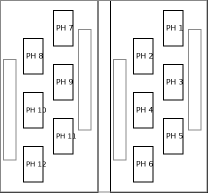
VISUALIZATION VISU_PhEnable_M2  // 208x193
    RoundedRectangle (0,0 98x193)
        toggle PRG_PRINT.sAdsPrintGroup[2].bI_Enable
    Rectangle (53,10 20x36), colour toggle: PRG_PRINT.sAdsPrintHead[7].bI_Enable
        toggle PRG_PRINT.sAdsPrintHead[7].bI_Enable
    Rectangle (23,38 20x36), colour toggle: PRG_PRINT.sAdsPrintHead[8].bI_Enable
        toggle PRG_PRINT.sAdsPrintHead[8].bI_Enable
    Rectangle (53,64 20x36), colour toggle: PRG_PRINT.sAdsPrintHead[9].bI_Enable
        toggle PRG_PRINT.sAdsPrintHead[9].bI_Enable
    Rectangle (23,92 20x36), colour toggle: PRG_PRINT.sAdsPrintHead[10].bI_Enable
        toggle PRG_PRINT.sAdsPrintHead[10].bI_Enable
    Rectangle (53,118 20x36), colour toggle: PRG_PRINT.sAdsPrintHead[11].bI_Enable
        toggle PRG_PRINT.sAdsPrintHead[11].bI_Enable
    Rectangle (23,146 20x36), colour toggle: PRG_PRINT.sAdsPrintHead[12].bI_Enable
        toggle PRG_PRINT.sAdsPrintHead[12].bI_Enable
    Rectangle (15,46 36x20), angle 270, "PH 8", colour toggle: PRG_PRINT.sAdsPrintHead[8].bI_Enable
    Rectangle (45,18 36x20), angle 270, "PH 7", colour toggle: PRG_PRINT.sAdsPrintHead[7].bI_Enable
    Rectangle (45,72 36x20), angle 270, "PH 9", colour toggle: PRG_PRINT.sAdsPrintHead[9].bI_Enable
    Rectangle (15,100 36x20), angle 270, "PH 10", colour toggle: PRG_PRINT.sAdsPrintHead[10].bI_Enable
    Rectangle (45,126 36x20), angle 270, "PH 11", colour toggle: PRG_PRINT.sAdsPrintHead[11].bI_Enable
    Rectangle (15,154 36x20), angle 270, "PH 12", colour toggle: PRG_PRINT.sAdsPrintHead[12].bI_Enable
    Frame (78,29 13x101)
        shows _VISU_PcMiniVertical(m_Inst := PRG_PRINT.FB_PC[3])
    Frame (3,59 13x101)
        shows _VISU_PcMiniVertical(m_Inst := PRG_PRINT.FB_PC[4])
    RoundedRectangle (110,0 98x193)
        toggle PRG_PRINT.sAdsPrintGroup[1].bI_Enable
    Rectangle (163,10 20x36), colour toggle: PRG_PRINT.sAdsPrintHead[1].bI_Enable
        toggle PRG_PRINT.sAdsPrintHead[1].bI_Enable
    Rectangle (133,38 20x36), colour toggle: PRG_PRINT.sAdsPrintHead[2].bI_Enable
        toggle PRG_PRINT.sAdsPrintHead[2].bI_Enable
    Rectangle (163,64 20x36), colour toggle: PRG_PRINT.sAdsPrintHead[3].bI_Enable
        toggle PRG_PRINT.sAdsPrintHead[3].bI_Enable
    Rectangle (133,92 20x36), colour toggle: PRG_PRINT.sAdsPrintHead[4].bI_Enable
        toggle PRG_PRINT.sAdsPrintHead[4].bI_Enable
    Rectangle (163,118 20x36), colour toggle: PRG_PRINT.sAdsPrintHead[5].bI_Enable
        toggle PRG_PRINT.sAdsPrintHead[5].bI_Enable
    Rectangle (133,146 20x36), colour toggle: PRG_PRINT.sAdsPrintHead[6].bI_Enable
        toggle PRG_PRINT.sAdsPrintHead[6].bI_Enable
    Rectangle (125,46 36x20), angle 270, "PH 2"
    Rectangle (155,18 36x20), angle 270, "PH 1"
    Rectangle (155,72 36x20), angle 270, "PH 3"
    Rectangle (125,100 36x20), angle 270, "PH 4"
    Rectangle (155,126 36x20), angle 270, "PH 5"
    Rectangle (125,154 36x20), angle 270, "PH 6"
    Frame (188,29 13x101)
        shows _VISU_PcMiniVertical(m_Inst := PRG_PRINT.FB_PC[1])
    Frame (113,59 13x101)
        shows _VISU_PcMiniVertical(m_Inst := PRG_PRINT.FB_PC[2])
END_VISUALIZATION

(* stored: Version 1.1.0.1, ProductVersion 3.1.4024.9
   Visu VISU_PhEnable_M2: Id {d729b797-a6c2-45a8-b0bb-a221c2872dd1} *)
